(* PLC project LD_COMPLEX_1.project, Inovance company InoProShop(V1.9.0.1) InoProShop(V1.9.0.1) *)
(* stored: creationDateTime 2025-04-08T16:35:22.9552253, modificationDateTime 2025-04-08T16:20:58.5952028 *)

PROGRAM PLC_PRG
  VAR
    X_EN : BOOL;
    X_RstEn : BOOL;
    X_RstStart : BOOL;
    X_TrnOrgS : BOOL;
    X_LLftOrgS : BOOL;
    X_LClmpOrgS : BOOL;
    X_LClmpMovS : BOOL;
    X_LRotOrgS : BOOL;
    Y_ENO : BOOL;
    Y_Rsting : BOOL;
    Y_RstDone : BOOL;
    Y_TrnCylR : BOOL;
    Y_LLftCylR : BOOL;
    Y_LClmpCylR : BOOL;
    Y_LClmpCylM : BOOL;
    Y_LRotCylR : BOOL;
    XY_LClmpWM : BOOL;
    PLS_0 : R_TRIG;
    RstStep : INT;
  END_VAR
  VAR  (* added by the conversion: wires and edge detectors of the diagram *)
    _EQ22_ENO : BOOL;
    _EQ22_OUT : BOOL;
    _EQ35_ENO : BOOL;
    _EQ35_OUT : BOOL;
    _EQ43_ENO : BOOL;
    _EQ43_OUT : BOOL;
    _EQ64_ENO : BOOL;
    _EQ64_OUT : BOOL;
    _EQ74_ENO : BOOL;
    _EQ74_OUT : BOOL;
  END_VAR

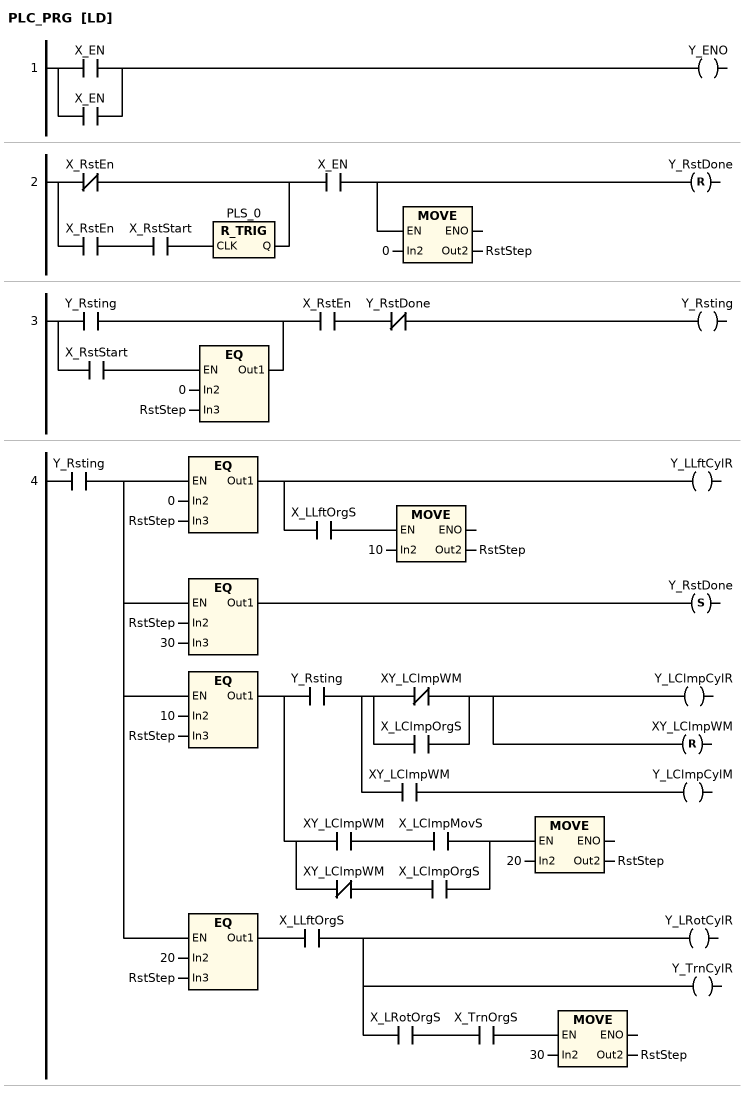
(* LD diagram, written out as Structured Text *)
(* 网络注释 *)

Y_ENO := X_EN;
(* 网络注释 *)

PLS_0(CLK := X_RstEn AND X_RstStart);
IF (NOT X_RstEn OR PLS_0.Q) AND X_EN THEN Y_RstDone := FALSE; END_IF;
IF (NOT X_RstEn OR PLS_0.Q) AND X_EN THEN RstStep := 0; END_IF;
(* 网络注释 *)

_EQ22_OUT := EQ(EN := X_RstStart, IN1 := 0, IN2 := RstStep, ENO => _EQ22_ENO);
Y_Rsting := (_EQ22_OUT OR Y_Rsting) AND X_RstEn AND NOT Y_RstDone;
(* 网络注释 *)

_EQ35_OUT := EQ(EN := Y_Rsting, IN1 := 0, IN2 := RstStep, ENO => _EQ35_ENO);
Y_LLftCylR := _EQ35_OUT;
IF _EQ35_OUT AND X_LLftOrgS THEN RstStep := 10; END_IF;
_EQ43_OUT := EQ(EN := Y_Rsting, IN1 := 10, IN2 := RstStep, ENO => _EQ43_ENO);
Y_LClmpCylR := _EQ43_OUT AND Y_Rsting AND (NOT XY_LClmpWM OR X_LClmpOrgS);
IF _EQ43_OUT AND Y_Rsting AND (NOT XY_LClmpWM OR X_LClmpOrgS) THEN XY_LClmpWM := FALSE; END_IF;
Y_LClmpCylM := _EQ43_OUT AND Y_Rsting AND XY_LClmpWM;
IF _EQ43_OUT AND (XY_LClmpWM AND X_LClmpMovS OR NOT XY_LClmpWM AND X_LClmpOrgS) THEN RstStep := 20; END_IF;
_EQ64_OUT := EQ(EN := Y_Rsting, IN1 := 20, IN2 := RstStep, ENO => _EQ64_ENO);
Y_LRotCylR := _EQ64_OUT AND X_LLftOrgS;
Y_TrnCylR := _EQ64_OUT AND X_LLftOrgS;
IF _EQ64_OUT AND X_LLftOrgS AND X_LRotOrgS AND X_TrnOrgS THEN RstStep := 30; END_IF;
_EQ74_OUT := EQ(EN := Y_Rsting, IN1 := RstStep, IN2 := 30, ENO => _EQ74_ENO);
IF _EQ74_OUT THEN Y_RstDone := TRUE; END_IF;
END_PROGRAM
